Fanuc KAREL source: kc00030.KL

-- PROVISIONAL review KL for V940-1; original PC SHA256 83d99be5673624494d4db72410d5718e23bed4d95c1d0e48b8a55305c877e1fb
-- Incomplete behavior may be omitted. Consult companion uncertainty JSON. Do not deploy.
PROGRAM KC00030
%NOLOCKGROUP
BEGIN
  -- V9_ZERO_TABLE_METADATA_HINT layout=0002_ascii; no indexed target words; source/name/runtime held
  -- UNRESOLVED_PC offsets 5-17; opcodes 3F,75
  -- UNRESOLVED_PC offsets 22-94; opcodes 27,22,2A,22,22,22,22,22,22,22,22,22,22,31
  -- UNRESOLVED_PC offsets 99-103; opcodes 7F
END KC00030
